{attribute 'qualified_only'}
TYPE E_CoeState :
(
    Init := 0,
    Read,
    ReadPeriodically,
    Error,
    Idle,
    PreRead,
    Calculate
);
END_TYPE

(* stored: Version 1.1.0.1, ProductVersion 3.1.4022.18
   DUT E_CoeState: Id {152610e0-cdbf-4e25-93df-dac94cd9b39b} *)
